    rq_wait_ft_sensor_steady(2000)
    zero_ftsensor()
    sleep(0.1)
    # end: URCap Program Node
    $ 100 "MoveL"
    $ 101 "ready_left" "breakAfter"
    set_tcp(p[0.00318,0.11464,0.09820000000000001,-0.7853981633974483,0.0,0.0])
    movel(pose_trans(CubeFront, pose_trans(p[-.002001169423, -.178123008725, .618090231485, -1.568699287997, .013964727372, .007428573496], ready_left_p)), a=1.2, v=0.25)
    # begin: URCap Program Node
    #   Source: Robotiq_Copilot, 1.22.1.14215, Robotiq Inc.
    #   Type: Find Surface
    $ 102 "Find Surface"
    zero_ftsensor()
    sleep(0.1)
    surface_found = rq_linear_search_urcap("Z+", 10.000, 0.005000, 0.100000, 1)
    storevar.setvariablepose("rq_findSurface_4ad0327a-680b-4db6-9ca5-7d81c97739c5_exitPosition", get_actual_tcp_pose())
    $ 103 "'Add Stop conditions from the Find Surface node'" "noBreak"
    # 'Add Stop conditions from the Find Surface node'
    # end: URCap Program Node
    # begin: URCap Program Node
    #   Source: Robotiq_Copilot, 1.22.1.14215, Robotiq Inc.
    #   Type: Finishing Tool Control
    $ 104 "Start tool"
    set_standard_digital_out(0, True)
    # end: URCap Program Node
    $ 105 "Wait: 0.5"
    sleep(0.5)
    $ 106 "Force"
    sleep(0.02)
    zero_ftsensor()
    force_mode(tool_pose(), [0, 0, 1, 0, 0, 0], [0.0, 0.0, 5.0, 0.0, 0.0, 0.0], 2, [0.1, 0.1, 0.15, 0.3490658503988659, 0.3490658503988659, 0.3490658503988659])
    $ 107 "Waypoint_44" "noBreak"
    set_tcp(p[0.00318,0.11464,0.09820000000000001,-0.7853981633974483,0.0,0.0])
    movel(pose_trans(CubeFront, pose_trans(p[-.084982669378, -.190534358862, .655595398108, -1.570665135698, -.001004032290, .001222209979], Waypoint_44_p)), a=1.2, v=0.05)
    end_force_mode()
    stopl(5.0)
    # begin: URCap Program Node
    #   Source: Robotiq_Copilot, 1.22.1.14215, Robotiq Inc.
    #   Type: Finishing Tool Control
    $ 108 "Stop tool"
    set_standard_digital_out(0, False)
    # end: URCap Program Node
    $ 109 "Waypoint_4" "breakAfter"
    set_tcp(p[0.00318,0.11464,0.09820000000000001,-0.7853981633974483,0.0,0.0])
    movel(pose_trans(CubeFront, pose_trans(p[-.084982669378, -.190534358862, .655595398108, -1.570665135698, -.001004032290, .001222209979], Waypoint_4_p)), a=1.2, v=0.25)
    $ 110 "clear" "breakAfter"
    set_tcp(p[0.00318,0.11464,0.09820000000000001,-0.7853981633974483,0.0,0.0])
    movel(pose_trans(CubeFront, pose_trans(p[.011052418258, -.164637958044, .620034439816, -1.578146963561, .014102050279, .014132657073], clear_p)), a=1.2, v=0.25)
    $ 111 "Waypoint_2" "breakAfter"
    set_tcp(p[0.00318,0.11464,0.09820000000000001,-0.7853981633974483,0.0,0.0])
    movel(pose_trans(CubeFront, pose_trans(p[-.005597006121, -.192408094989, .653246871754, -1.571622694982, -.002967386491, .002471774867], Waypoint_2_p)), a=1.2, v=0.25)
    $ 112 "Waypoint_3" "breakAfter"
    set_tcp(p[0.00318,0.11464,0.09820000000000001,-0.7853981633974483,0.0,0.0])
    movel(pose_trans(CubeFront, pose_trans(p[-.002001169423, -.178123008725, .618090231485, -1.568699287997, .013964727372, .007428573496], Waypoint_3_p)), a=1.2, v=0.25)
    # begin: URCap Program Node
    #   Source: Robotiq_Copilot, 1.22.1.14215, Robotiq Inc.
    #   Type: Find Surface
    $ 113 "Find Surface"
    zero_ftsensor()
    sleep(0.1)
    surface_found = rq_linear_search_urcap("Z+", 10.000, 0.005000, 0.100000, 1)
    storevar.setvariablepose("rq_findSurface_a4bee10f-93fa-4f90-9b91-ae0c246f4091_exitPosition", get_actual_tcp_pose())
    $ 114 "'Add Stop conditions from the Find Surface node'" "noBreak"
    # 'Add Stop conditions from the Find Surface node'
    # end: URCap Program Node
    # begin: URCap Program Node
    #   Source: Robotiq_Copilot, 1.22.1.14215, Robotiq Inc.
    #   Type: Finishing Tool Control
    $ 115 "Start tool"
    set_standard_digital_out(0, True)
    # end: URCap Program Node
    $ 116 "Wait: 0.5"
    sleep(0.5)
    $ 117 "Force"
    sleep(0.02)
    zero_ftsensor()
    force_mode(tool_pose(), [0, 0, 1, 0, 0, 0], [0.0, 0.0, 5.0, 0.0, 0.0, 0.0], 2, [0.1, 0.1, 0.15, 0.3490658503988659, 0.3490658503988659, 0.3490658503988659])
    $ 118 "Waypoint_8" "noBreak"
    set_tcp(p[0.00318,0.11464,0.09820000000000001,-0.7853981633974483,0.0,0.0])
    movel(pose_trans(CubeFront, pose_trans(p[-.002001169423, -.178123008725, .618090231485, -1.568699287997, .013964727372, .007428573496], Waypoint_8_p)), a=1.2, v=0.05)
    $ 119 "Waypoint_5" "noBreak"
    set_tcp(p[0.00318,0.11464,0.09820000000000001,-0.7853981633974483,0.0,0.0])
    movel(pose_trans(CubeFront, pose_trans(p[-.002001169423, -.178123008725, .618090231485, -1.568699287997, .013964727372, .007428573496], Waypoint_5_p)), a=1.2, v=0.05)
    end_force_mode()
    stopl(5.0)
    # begin: URCap Program Node
    #   Source: Robotiq_Copilot, 1.22.1.14215, Robotiq Inc.
    #   Type: Finishing Tool Control
    $ 120 "Stop tool"
    set_standard_digital_out(0, False)
    # end: URCap Program Node
    $ 121 "Waypoint_17" "breakAfter"
    set_tcp(p[0.00318,0.11464,0.09820000000000001,-0.7853981633974483,0.0,0.0])
    movel(pose_trans(CubeFront, pose_trans(p[-.005597006121, -.192408094989, .653246871754, -1.571622694982, -.002967386491, .002471774867], Waypoint_17_p)), a=1.2, v=0.25)
    $ 122 "MoveJ"
    $ 123 "Waypoint_11" "breakAfter"
    movej(get_inverse_kin(pose_trans(CubeFront, pose_trans(p[-.005597006121, -.192408094989, .653246871754, -1.571622694982, -.002967386491, .002471774867], Waypoint_11_p)), qnear=Waypoint_11_q), a=1.3962634015954636, v=1.0471975511965976)
    $ 124 "Waypoint_6" "breakAfter"
    movej(get_inverse_kin(pose_trans(CubeFront, pose_trans(p[-.005597006121, -.192408094989, .653246871754, -1.571622694982, -.002967386491, .002471774867], Waypoint_6_p)), qnear=Waypoint_6_q), a=1.3962634015954636, v=1.0471975511965976)
    $ 125 "Waypoint_31" "breakAfter"
    movej(get_inverse_kin(pose_trans(CubeFront, pose_trans(p[-.002001169423, -.178123008725, .618090231485, -1.568699287997, .013964727372, .007428573496], Waypoint_31_p)), qnear=Waypoint_31_q), a=1.3962634015954636, v=1.0471975511965976)
    # begin: URCap Program Node
    #   Source: Robotiq_Copilot, 1.22.1.14215, Robotiq Inc.
    #   Type: Zero FT Sensor
    $ 126 "Zero FT Sensor"

    rq_wait_ft_sensor_steady(2000)
    zero_ftsensor()
    sleep(0.1)
    # end: URCap Program Node
    # begin: URCap Program Node
    #   Source: Robotiq_Copilot, 1.22.1.14215, Robotiq Inc.
    #   Type: Find Surface
    $ 127 "Find Surface"
    zero_ftsensor()
    sleep(0.1)
    surface_found = rq_linear_search_urcap("Z+", 10.000, 0.005000, 0.100000, 1)
    storevar.setvariablepose("rq_findSurface_84b4ea62-5d9f-42a8-b409-36e608cbcae1_exitPosition", get_actual_tcp_pose())
    $ 128 "'Add Stop conditions from the Find Surface node'" "noBreak"
    # 'Add Stop conditions from the Find Surface node'
    # end: URCap Program Node
    # begin: URCap Program Node
    #   Source: Robotiq_Copilot, 1.22.1.14215, Robotiq Inc.
    #   Type: Finishing Tool Control
    $ 129 "Start tool"
    set_standard_digital_out(0, True)
    # end: URCap Program Node
    $ 130 "Wait: 0.5"
    sleep(0.5)
    $ 131 "Force"
    sleep(0.02)
    zero_ftsensor()
    force_mode(tool_pose(), [0, 0, 1, 0, 0, 0], [0.0, 0.0, 5.0, 0.0, 0.0, 0.0], 2, [0.1, 0.1, 0.15, 0.3490658503988659, 0.3490658503988659, 0.3490658503988659])
    $ 132 "Waypoint_7" "noBreak"
    set_tcp(p[0.00318,0.11464,0.09820000000000001,-0.7853981633974483,0.0,0.0])
    movel(pose_trans(CubeFront, pose_trans(p[-.005597006121, -.192408094989, .653246871754, -1.571622694982, -.002967386491, .002471774867], Waypoint_7_p)), a=1.2, v=0.05)
    end_force_mode()
    stopl(5.0)
    # begin: URCap Program Node
    #   Source: Robotiq_Copilot, 1.22.1.14215, Robotiq Inc.
    #   Type: Finishing Tool Control
    $ 133 "Stop tool"
    set_standard_digital_out(0, False)
    # end: URCap Program Node
    $ 134 "Waypoint_13" "breakAfter"
    set_tcp(p[0.00318,0.11464,0.09820000000000001,-0.7853981633974483,0.0,0.0])
    movel(pose_trans(CubeFront, pose_trans(p[-.002001169423, -.178123008725, .618090231485, -1.568699287997, .013964727372, .007428573496], Waypoint_13_p)), a=1.2, v=0.25)
    $ 135 "Waypoint_9" "breakAfter"
    set_tcp(p[0.00318,0.11464,0.09820000000000001,-0.7853981633974483,0.0,0.0])
    movel(pose_trans(CubeFront, pose_trans(p[-.002001169423, -.178123008725, .618090231485, -1.568699287997, .013964727372, .007428573496], Waypoint_9_p)), a=1.2, v=0.25)
    $ 136 "clear" "breakAfter"
    set_tcp(p[0.00318,0.11464,0.09820000000000001,-0.7853981633974483,0.0,0.0])
    movel(pose_trans(CubeFront, pose_trans(p[.011052418258, -.164637958044, .620034439816, -1.578146963561, .014102050279, .014132657073], clear_p)), a=1.2, v=0.25)
  end
  def SprayFront():
    $ 137 "SprayFront" "noBreak"
    $ 138 "SprayFront"
    $ 139 "MoveJ"
    $ 140 "clear" "breakAfter"
    set_tcp(p[0.00318,0.11464,0.09820000000000001,-0.7853981633974483,0.0,0.0])
    movej(get_inverse_kin(pose_trans(CubeFront, pose_trans(p[.011052418258, -.164637958044, .620034439816, -1.578146963561, .014102050279, .014132657073], clear_p)), qnear=clear_q), a=1.3962634015954636, v=1.0471975511965976)
    $ 141 "MoveJ"
    $ 142 "Waypoint_10" "breakAfter"
    set_tcp(p[0.020839023181949995,-0.027139950822234082,0.10599373590389219,0.12258870209179472,1.1769383890382668,2.869747076630172])
    movej(get_inverse_kin(pose_trans(CubeFront, pose_trans(p[-.002001169423, -.178123008725, .618090231485, -1.568699287997, .013964727372, .007428573496], Waypoint_10_p)), qnear=Waypoint_10_q), a=1.3962634015954636, v=1.0471975511965976)
    $ 143 "Set DO[1]=On"
    set_standard_digital_out(1, True)
    $ 144 "MoveL"
    $ 145 "Waypoint_12" "breakAfter"
    movel(pose_trans(CubeFront, pose_trans(p[-.002001169423, -.178123008725, .618090231485, -1.568699287997, .013964727372, .007428573496], Waypoint_12_p)), a=1.2, v=0.1)
    $ 146 "Set DO[1]=Off"
    set_standard_digital_out(1, False)
    $ 147 "MoveJ"
    $ 148 "Waypoint_21" "breakAfter"
    set_tcp(p[0.020839023181949995,-0.027139950822234082,0.10599373590389219,0.12258870209179472,1.1769383890382668,2.869747076630172])
    movej(get_inverse_kin(pose_trans(CubeFront, pose_trans(p[-.002001169423, -.178123008725, .618090231485, -1.568699287997, .013964727372, .007428573496], Waypoint_21_p)), qnear=Waypoint_21_q), a=1.3962634015954636, v=1.0471975511965976)
    $ 149 "Set DO[1]=On"
    set_standard_digital_out(1, True)
    $ 150 "MoveL"
    $ 151 "Waypoint_22" "breakAfter"
    set_tcp(p[0.020839023181949995,-0.027139950822234082,0.10599373590389219,0.12258870209179472,1.1769383890382668,2.869747076630172])
    movel(pose_trans(CubeFront, pose_trans(p[-.002001169423, -.178123008725, .618090231485, -1.568699287997, .013964727372, .007428573496], Waypoint_22_p)), a=1.2, v=0.1)
    $ 152 "Set DO[1]=Off"
    set_standard_digital_out(1, False)
    $ 153 "MoveJ"
    $ 154 "Waypoint_23" "breakAfter"
    set_tcp(p[0.020839023181949995,-0.027139950822234082,0.10599373590389219,0.12258870209179472,1.1769383890382668,2.869747076630172])
    movej(get_inverse_kin(pose_trans(CubeFront, pose_trans(p[-.002001169423, -.178123008725, .618090231485, -1.568699287997, .013964727372, .007428573496], Waypoint_23_p)), qnear=Waypoint_23_q), a=1.3962634015954636, v=1.0471975511965976)
    $ 155 "Set DO[1]=On"
    set_standard_digital_out(1, True)
    $ 156 "MoveL"
    $ 157 "Waypoint_24" "breakAfter"
    set_tcp(p[0.020839023181949995,-0.027139950822234082,0.10599373590389219,0.12258870209179472,1.1769383890382668,2.869747076630172])
    movel(pose_trans(CubeFront, pose_trans(p[-.002001169423, -.178123008725, .618090231485, -1.568699287997, .013964727372, .007428573496], Waypoint_24_p)), a=1.2, v=0.1)
    $ 158 "Set DO[1]=Off"
    set_standard_digital_out(1, False)
    $ 159 "MoveJ"
    $ 160 "clear" "breakAfter"
    movej(clear_q, a=1.3962634015954636, v=1.0471975511965976)
    $ 161 "MoveJ"
    $ 162 "Waypoint_26" "breakAfter"
    set_tcp(p[0.020839023181949995,-0.027139950822234082,0.10599373590389219,0.12258870209179472,1.1769383890382668,2.869747076630172])
    movej(get_inverse_kin(pose_trans(CubeFront, pose_trans(p[-.002001169423, -.178123008725, .618090231485, -1.568699287997, .013964727372, .007428573496], Waypoint_26_p)), qnear=Waypoint_26_q), a=1.3962634015954636, v=1.0471975511965976)
    $ 163 "Set DO[1]=On"
    set_standard_digital_out(1, True)
    $ 164 "MoveL"
    $ 165 "Waypoint_25" "breakAfter"
    set_tcp(p[0.020839023181949995,-0.027139950822234082,0.10599373590389219,0.12258870209179472,1.1769383890382668,2.869747076630172])
    movel(pose_trans(CubeFront, pose_trans(p[-.002001169423, -.178123008725, .618090231485, -1.568699287997, .013964727372, .007428573496], Waypoint_25_p)), a=1.2, v=0.1)
    $ 166 "Set DO[1]=Off"
    set_standard_digital_out(1, False)
    $ 167 "MoveJ"
    $ 168 "clear" "breakAfter"
    movej(clear_q, a=1.3962634015954636, v=1.0471975511965976)
  end
  def SprayRebate():
    $ 169 "SprayRebate" "noBreak"
    $ 170 "SprayRebate"
    $ 171 "MoveJ"
    $ 172 "clear" "breakAfter"
    movej(clear_q, a=1.3962634015954636, v=1.0471975511965976)
    $ 173 "MoveJ"
    $ 174 "Waypoint_28" "breakAfter"
    set_tcp(p[0.020839023181949995,-0.027139950822234082,0.10599373590389219,0.12258870209179472,1.1769383890382668,2.869747076630172])
    movej(get_inverse_kin(pose_trans(CubeFront, pose_trans(p[-.002001169423, -.178123008725, .618090231485, -1.568699287997, .013964727372, .007428573496], Waypoint_28_p)), qnear=Waypoint_28_q), a=1.3962634015954636, v=1.0471975511965976)
    $ 175 "Set DO[1]=On"
    set_standard_digital_out(1, True)
    $ 176 "MoveL"
    $ 177 "Waypoint_27" "breakAfter"
    set_tcp(p[0.020839023181949995,-0.027139950822234082,0.10599373590389219,0.12258870209179472,1.1769383890382668,2.869747076630172])
    movel(pose_trans(CubeFront, pose_trans(p[-.002001169423, -.178123008725, .618090231485, -1.568699287997, .013964727372, .007428573496], Waypoint_27_p)), a=1.2, v=0.1)
    $ 178 "Set DO[1]=Off"
    set_standard_digital_out(1, False)
    $ 179 "MoveJ"
    $ 180 "Waypoint_29" "breakAfter"
    set_tcp(p[0.020839023181949995,-0.027139950822234082,0.10599373590389219,0.12258870209179472,1.1769383890382668,2.869747076630172])
    movej(get_inverse_kin(pose_trans(CubeFront, pose_trans(p[-.002001169423, -.178123008725, .618090231485, -1.568699287997, .013964727372, .007428573496], Waypoint_29_p)), qnear=Waypoint_29_q), a=1.3962634015954636, v=1.0471975511965976)
    $ 181 "Set DO[1]=On"
    set_standard_digital_out(1, True)
    $ 182 "MoveL"
    $ 183 "Waypoint_30" "breakAfter"
    set_tcp(p[0.020839023181949995,-0.027139950822234082,0.10599373590389219,0.12258870209179472,1.1769383890382668,2.869747076630172])
    movel(pose_trans(CubeFront, pose_trans(p[-.002001169423, -.178123008725, .618090231485, -1.568699287997, .013964727372, .007428573496], Waypoint_30_p)), a=1.2, v=0.1)
    $ 184 "Set DO[1]=Off"
    set_standard_digital_out(1, False)
    $ 185 "MoveJ"
    $ 186 "clear" "breakAfter"
    movej(clear_q, a=1.3962634015954636, v=1.0471975511965976)
    $ 187 "MoveJ"
    $ 188 "Waypoint_32" "breakAfter"
    set_tcp(p[0.020839023181949995,-0.027139950822234082,0.10599373590389219,0.12258870209179472,1.1769383890382668,2.869747076630172])
    movej(get_inverse_kin(pose_trans(CubeFront, pose_trans(p[-.002001169423, -.178123008725, .618090231485, -1.568699287997, .013964727372, .007428573496], Waypoint_32_p)), qnear=Waypoint_32_q), a=1.3962634015954636, v=1.0471975511965976)
    $ 189 "Set DO[1]=On"
    set_standard_digital_out(1, True)
    $ 190 "MoveL"
    $ 191 "Waypoint_33" "breakAfter"
    set_tcp(p[0.020839023181949995,-0.027139950822234082,0.10599373590389219,0.12258870209179472,1.1769383890382668,2.869747076630172])
    movel(pose_trans(CubeFront, pose_trans(p[-.002001169423, -.178123008725, .618090231485, -1.568699287997, .013964727372, .007428573496], Waypoint_33_p)), a=1.2, v=0.1)
    $ 192 "Set DO[1]=Off"
    set_standard_digital_out(1, False)
    $ 193 "MoveJ"
    $ 194 "clear" "breakAfter"
    movej(clear_q, a=1.3962634015954636, v=1.0471975511965976)
  end
  def SandFront():
    $ 195 "SandFront" "noBreak"
    $ 196 "sandFront"
    $ 197 "MoveL"
    $ 198 "Waypoint_1" "breakAfter"
    set_tcp(p[0.00318,0.11464,0.09820000000000001,-0.7853981633974483,0.0,0.0])
    movel(pose_trans(WorkPlane, pose_trans(p[-.005597006121, -.192408094989, .653246871754, -1.571622694982, -.002967386491, .002471774867], Waypoint_1_p)), a=1.2, v=0.25)
    # begin: URCap Program Node
    #   Source: Robotiq_Copilot, 1.22.1.14215, Robotiq Inc.
    #   Type: Zero FT Sensor
    $ 199 "Zero FT Sensor"

    rq_wait_ft_sensor_steady(2000)
    zero_ftsensor()
    sleep(0.1)
    # end: URCap Program Node
    # begin: URCap Program Node
    #   Source: Robotiq_Copilot, 1.22.1.14215, Robotiq Inc.
    #   Type: Find Surface
    $ 200 "Find Surface"
    surface_found = rq_linear_search_urcap("Z+", 10.000, 0.005000, 0.100000, 1)
    storevar.setvariablepose("rq_findSurface_05849863-69e7-4f05-b7d8-49d959ee6416_exitPosition", get_actual_tcp_pose())
    $ 201 "'Add Stop conditions from the Find Surface node'" "noBreak"
    # 'Add Stop conditions from the Find Surface node'
    # end: URCap Program Node
    # begin: URCap Program Node
    #   Source: Robotiq_Copilot, 1.22.1.14215, Robotiq Inc.
    #   Type: Finishing Tool Control
    $ 202 "Start tool"
    set_standard_digital_out(0, True)
    # end: URCap Program Node
    $ 203 "Wait: 0.5"
    sleep(0.5)
    $ 204 "MoveL"
    $ 205 "Force"
    sleep(0.02)
    zero_ftsensor()
    force_mode(tool_pose(), [0, 0, 1, 0, 0, 0], [0.0, 0.0, 5.0, 0.0, 0.0, 0.0], 2, [0.1, 0.1, 0.15, 0.3490658503988659, 0.3490658503988659, 0.3490658503988659])
    $ 206 "Waypoint_35" "noBreak"
    set_tcp(p[0.00318,0.11464,0.09820000000000001,-0.7853981633974483,0.0,0.0])
    movel(pose_trans(WorkPlane, pose_trans(p[.011052418258, -.164637958044, .620034439816, -1.578146963561, .014102050279, .014132657073], Waypoint_35_p)), a=1.2, v=0.06)
    $ 207 "Waypoint_36" "noBreak"
    set_tcp(p[0.00318,0.11464,0.09820000000000001,-0.7853981633974483,0.0,0.0])
    movel(pose_trans(WorkPlane, pose_trans(p[.011052418258, -.164637958044, .620034439816, -1.578146963561, .014102050279, .014132657073], Waypoint_36_p)), a=1.2, v=0.06)
    $ 208 "Waypoint_37" "noBreak"
    set_tcp(p[0.00318,0.11464,0.09820000000000001,-0.7853981633974483,0.0,0.0])
    movel(pose_trans(WorkPlane, pose_trans(p[.011052418258, -.164637958044, .620034439816, -1.578146963561, .014102050279, .014132657073], Waypoint_37_p)), a=1.2, v=0.06)
    $ 209 "Waypoint_38" "noBreak"
    set_tcp(p[0.00318,0.11464,0.09820000000000001,-0.7853981633974483,0.0,0.0])
    movel(pose_trans(WorkPlane, pose_trans(p[.011052418258, -.164637958044, .620034439816, -1.578146963561, .014102050279, .014132657073], Waypoint_38_p)), a=1.2, v=0.06)
    # begin: URCap Program Node
    #   Source: Robotiq_Copilot, 1.22.1.14215, Robotiq Inc.
    #   Type: Finishing Tool Control
    $ 210 "Stop tool" "noBreak"
    set_standard_digital_out(0, False)
    # end: URCap Program Node
    end_force_mode()
    stopl(5.0)
    $ 211 "Direction: Tool Z-"
    global move_thread_flag_211=0
    thread move_thread_211():
      enter_critical
      move_thread_flag_211 = 1
      local towardsPos=calculate_point_to_move_towards(get_forward_kin(), [0.0,0.0,-1.0], 0.025)
      movel(towardsPos, a=1.2, v=0.06)
      move_thread_flag_211 = 2
      exit_critical
    end
    move_thread_flag_211 = 0
    move_thread_han_211 = run move_thread_211()
    while (True):
      sleep(1.0E-10)
      if (move_thread_flag_211 > 1):
        join move_thread_han_211
        $ 212 "Until (distance)"
        break
      end
      sync()
    end
  end
  def StartSpray():
    $ 213 "StartSpray" "noBreak"
    $ 214 "Set DO[1]=On"
    set_standard_digital_out(1, True)
    $ 215 "Wait: 0.3"
    sleep(0.3)
  end
  def stopSpray():
    $ 216 "stopSpray" "noBreak"
    $ 217 "Set DO[1]=Off"
    set_standard_digital_out(1, False)
    $ 218 "Wait: 0.3"
    sleep(0.3)
  end
  $ 1 "BeforeStart"
  $ 2 "WorkPlane≔CubeFront"
  global WorkPlane=CubeFront
  thread EventThread():
    while (True):
      if (get_standard_digital_in(1) !=   True  ):
        $ 92 "Set DO[0]=Off"
        set_standard_digital_out(0, False)
        $ 93 "Set DO[1]=Off"
        set_standard_digital_out(1, False)
        $ 94 "Halt"
        halt
      end
      sync()
    end
  end
  eventThread = run EventThread()
  $ 3 "Robot Program"
  $ 4 "Main"
  $ 5 "MoveJ"
  $ 6 "clear" "breakAfter"
  set_tcp(p[0.00318,0.11464,0.09820000000000001,-0.7853981633974483,0.0,0.0])
  movej(get_inverse_kin(pose_trans(CubeFront, pose_trans(p[.011052418258, -.164637958044, .620034439816, -1.578146963561, .014102050279, .014132657073], clear_p)), qnear=clear_q), a=1.3962634015954636, v=1.0471975511965976)
  # begin: URCap Program Node
  #   Source: Robotiq_Copilot, 1.22.1.14215, Robotiq Inc.
  #   Type: Zero FT Sensor
  $ 7 "Zero FT Sensor"

  rq_wait_ft_sensor_steady(2000)
  zero_ftsensor()
  sleep(0.1)
  # end: URCap Program Node
  $ 8 "WorkPlane≔CubeFront"
  global WorkPlane=CubeFront
  $ 9 "Call SandFront"
  SandFront()
  $ 10 "MoveJ"
  $ 11 "clear" "breakAfter"
  set_tcp(p[0.00318,0.11464,0.09820000000000001,-0.7853981633974483,0.0,0.0])
  movej(get_inverse_kin(pose_trans(CubeFront, pose_trans(p[.011052418258, -.164637958044, .620034439816, -1.578146963561, .014102050279, .014132657073], clear_p)), qnear=clear_q), a=1.3962634015954636, v=1.0471975511965976)
  # begin: URCap Program Node
  #   Source: Robotiq_Copilot, 1.22.1.14215, Robotiq Inc.
  #   Type: Zero FT Sensor
  $ 12 "Zero FT Sensor"

  rq_wait_ft_sensor_steady(2000)
  zero_ftsensor()
  sleep(0.1)
  # end: URCap Program Node
  $ 13 "Call ChamferFace"
  ChamferFace()
  $ 14 "MoveJ"
  $ 15 "clear" "breakAfter"
  set_tcp(p[0.00318,0.11464,0.09820000000000001,-0.7853981633974483,0.0,0.0])
  movej(get_inverse_kin(pose_trans(CubeFront, pose_trans(p[.011052418258, -.164637958044, .620034439816, -1.578146963561, .014102050279, .014132657073], clear_p)), qnear=clear_q), a=1.3962634015954636, v=1.0471975511965976)
  # begin: URCap Program Node
  #   Source: Robotiq_Copilot, 1.22.1.14215, Robotiq Inc.
  #   Type: Zero FT Sensor
  $ 16 "Zero FT Sensor"

  rq_wait_ft_sensor_steady(2000)
  zero_ftsensor()
  sleep(0.1)
  # end: URCap Program Node
  $ 17 "WorkPlane≔SandBack"
  global WorkPlane=SandBack
  $ 18 "MoveJ"
  $ 19 "clear" "breakAfter"
  set_tcp(p[0.00318,0.11464,0.09820000000000001,-0.7853981633974483,0.0,0.0])
  movej(get_inverse_kin(pose_trans(SandBack, pose_trans(p[.011052418258, -.164637958044, .620034439816, -1.578146963561, .014102050279, .014132657073], clear_p)), qnear=clear_q), a=1.3962634015954636, v=1.0471975511965976)
  # begin: URCap Program Node
  #   Source: Robotiq_Copilot, 1.22.1.14215, Robotiq Inc.
  #   Type: Zero FT Sensor
  $ 20 "Zero FT Sensor"

  rq_wait_ft_sensor_steady(2000)
  zero_ftsensor()
  sleep(0.1)
  # end: URCap Program Node
  $ 21 "Call SandFront"
  SandFront()
  $ 22 "MoveJ"
  $ 23 "clear" "breakAfter"
  set_tcp(p[0.00318,0.11464,0.09820000000000001,-0.7853981633974483,0.0,0.0])
  movej(get_inverse_kin(pose_trans(SandBack, pose_trans(p[.011052418258, -.164637958044, .620034439816, -1.578146963561, .014102050279, .014132657073], clear_p)), qnear=clear_q), a=1.3962634015954636, v=1.0471975511965976)
  # begin: URCap Program Node
  #   Source: Robotiq_Copilot, 1.22.1.14215, Robotiq Inc.
  #   Type: Zero FT Sensor
  $ 24 "Zero FT Sensor"

  rq_wait_ft_sensor_steady(2000)
  zero_ftsensor()
  sleep(0.1)
  # end: URCap Program Node
  $ 25 "Call ChamferFace"
  ChamferFace()
  $ 26 "MoveJ"
  $ 27 "clear" "breakAfter"
  set_tcp(p[0.00318,0.11464,0.09820000000000001,-0.7853981633974483,0.0,0.0])
  movej(get_inverse_kin(pose_trans(SandBack, pose_trans(p[.011052418258, -.164637958044, .620034439816, -1.578146963561, .014102050279, .014132657073], clear_p)), qnear=clear_q), a=1.3962634015954636, v=1.0471975511965976)
  # begin: URCap Program Node
  #   Source: Robotiq_Copilot, 1.22.1.14215, Robotiq Inc.
  #   Type: Zero FT Sensor
  $ 28 "Zero FT Sensor"

  rq_wait_ft_sensor_steady(2000)
  zero_ftsensor()
  sleep(0.1)
  # end: URCap Program Node
end
